INTERFACE I_Conveyor

PROPERTY IsRun : BOOL
GET
END_GET
END_PROPERTY

METHOD Start : BOOL
VAR_INPUT
END_VAR
END_METHOD

METHOD Stop : BOOL
VAR_INPUT
END_VAR
END_METHOD

END_INTERFACE

(* stored: Version 1.1.0.1, ProductVersion 3.1.4024.12
   Itf I_Conveyor: Id {1b61c57b-208a-4700-9861-5506ae1b73c9}
   Property IsRun: Id {161f9925-bbe5-43d4-b9b0-22c3e9542b0a}
   Get Get: Id {01dd5a43-617a-41a8-a033-4239150ea30f}
   Method Start: Id {774e16e0-9a09-4a57-9fd6-a97390433df2}
   Method Stop: Id {93596a68-d5c6-4094-9c20-5046fbf6f761} *)
